{attribute 'GeneratedUsingTerminal: EL5151-0000-0017'}
{attribute addProperty BoxType "EL5151-0000-0017"}
{attribute addProperty Id "Latch_C_validAT %I*BOOL1Latch_extern_validAT %I*BOOL1Set_counter_doneAT %I*BOOL1Extrapolation_stallAT %I*BOOL1Status_of_input_AAT %I*BOOL1Status_of_input_BAT %I*BOOL1Status_of_input_CAT %I*BOOL1Status_of_extern_latchAT %I*BOOL1Sync_ErrorAT %I*BOOL1TxPDO_ToggleAT %I*BOOL1Counter_valueAT %I*UDINT4Latch_valueAT %I*UDINT4"}
{attribute addProperty CRC "1444807711"}
{attribute addProperty Size "18"}
TYPE ENC_Inputs_561E041F :
STRUCT
	{attribute addProperty Name "Latch_C_valid"}
	Latch_C_valid AT %I* : BOOL;
	{attribute addProperty Name "Latch_extern_valid"}
	Latch_extern_valid AT %I* : BOOL;
	{attribute addProperty Name "Set_counter_done"}
	Set_counter_done AT %I* : BOOL;
	{attribute addProperty Name "Extrapolation_stall"}
	Extrapolation_stall AT %I* : BOOL;
	{attribute addProperty Name "Status_of_input_A"}
	Status_of_input_A AT %I* : BOOL;
	{attribute addProperty Name "Status_of_input_B"}
	Status_of_input_B AT %I* : BOOL;
	{attribute addProperty Name "Status_of_input_C"}
	Status_of_input_C AT %I* : BOOL;
	{attribute addProperty Name "Status_of_extern_latch"}
	Status_of_extern_latch AT %I* : BOOL;
	{attribute addProperty Name "Sync_Error"}
	Sync_Error AT %I* : BOOL;
	{attribute addProperty Name "TxPDO_Toggle"}
	TxPDO_Toggle AT %I* : BOOL;
	{attribute addProperty Name "Counter_value"}
	Counter_value AT %I* : UDINT;
	{attribute addProperty Name "Latch_value"}
	Latch_value AT %I* : UDINT;
END_STRUCT
END_TYPE

(* stored: Version 1.2.0.0, ProductVersion 3.1.4024.9
   DUT ENC_Inputs_561E041F: Id {342f0387-59fa-4c41-9bbe-587761bd7b77} *)
